(* IEC 61131-3 sources: pandora/pandora/aws-platform-main/aws-platform-main/test/Io, 6 files *)

(* ---- Digital.st ---- *)
USING Esab.Io.Mock;

USING AxUnit;

NAMESPACE Esab.Io.Test

    {TestFixture}
    {Category(IO)}
    CLASS DigitalInputTests
        VAR PRIVATE
            _value : BOOL;
            _input : DigitalInput;
            _changedHandler : DigitalInputChangedListenerMock;
        END_VAR

        {FixtureSetup}
        METHOD PUBLIC TestFixtureSetup
            ;
        END_METHOD

        {TestSetup}
        METHOD PUBLIC TestSetup
            _changedHandler.Id := UINT#0;
            _changedHandler.Value := FALSE;
            // Read two times to reset state.
            _input.Id := UINT#0;
            _input.Read(FALSE);
            _input.Read(FALSE);
        END_METHOD

        {Test}
        METHOD PUBLIC GetValue
            _input.Read(TRUE);
            Assert.Equal(_input.GetValue(), TRUE);
            _input.Read(FALSE);
            Assert.Equal(_input.GetValue(), FALSE);
        END_METHOD

        {Test}
        METHOD PUBLIC RisingEdge
            _input.Read(TRUE);
            Assert.Equal(_input.GetValue(), TRUE);
            Assert.Equal(_input.RisingEdge(), TRUE);
            Assert.Equal(_input.FallingEdge(), FALSE);
            _input.Read(TRUE);
            Assert.Equal(_input.GetValue(), TRUE);
            Assert.Equal(_input.RisingEdge(), FALSE);
            Assert.Equal(_input.FallingEdge(), FALSE);
        END_METHOD

        {Test}
        METHOD PUBLIC FallingEdge
            _input.Read(TRUE);
            Assert.Equal(_input.GetValue(), TRUE);
            _input.Read(FALSE);
            Assert.Equal(_input.GetValue(), FALSE);
            Assert.Equal(_input.RisingEdge(), FALSE);
            Assert.Equal(_input.FallingEdge(), TRUE);
            _input.Read(FALSE);
            Assert.Equal(_input.GetValue(), FALSE);
            Assert.Equal(_input.RisingEdge(), FALSE);
            Assert.Equal(_input.FallingEdge(), FALSE);
        END_METHOD

        {Test}
        METHOD PUBLIC OnChangedRising
            _input.Id := UINT#255;
            _input.SetChangedHandler(_changedHandler);

            _input.Read(FALSE);
            _input.Read(TRUE);

            Assert.Equal(_input.GetValue(), TRUE);
            Assert.Equal(_changedHandler.Id, UINT#255);
            Assert.Equal(_changedHandler.Value, TRUE);
        END_METHOD

        {Test}
        METHOD PUBLIC OnChangedFalling
            _input.Id := UINT#255;
            _input.SetChangedHandler(_changedHandler);

            _input.Read(FALSE);
            _input.Read(TRUE);
            _input.Read(FALSE);

            Assert.Equal(_input.GetValue(), FALSE);
            Assert.Equal(_changedHandler.Id, UINT#255);
            Assert.Equal(_changedHandler.Value, FALSE);
        END_METHOD

        {Test}
        METHOD PUBLIC HasChanged
            _input.Read(TRUE);
            _input.Read(TRUE);
            Assert.Equal(_input.HasChanged(), FALSE);
            _input.Read(FALSE);
            Assert.Equal(_input.HasChanged(), TRUE);
            _input.Read(TRUE);
            Assert.Equal(_input.HasChanged(), TRUE);
        END_METHOD
    END_CLASS

    {TestFixture}
    CLASS DigitalOutputTests
        VAR PRIVATE
            _outputValue : BOOL;
            _output : DigitalOutput;
        END_VAR

        {FixtureSetup}
        METHOD PUBLIC TestFixtureSetup
            ;
        END_METHOD

        {TestSetup}
        METHOD PUBLIC TestSetup
            _outputValue := FALSE;
            _output.SetValue(_outputValue);
        END_METHOD

        {Test}
        METHOD PUBLIC Set
            _output.Set();
            _output.Write(value => _outputValue);

            Assert.Equal(_outputValue, TRUE);
        END_METHOD

        {Test}
        METHOD PUBLIC Reset
            _outputValue := TRUE;
            _output.Reset();
            _output.Write(value => _outputValue);

            Assert.Equal(_outputValue, FALSE);
        END_METHOD

        {Test}
        METHOD PUBLIC Toggle
            _output.Toggle();
            _output.Write(value => _outputValue);

            Assert.Equal(_outputValue, TRUE);

            _output.Toggle();
            _output.Write(value => _outputValue);

            Assert.Equal(_outputValue, FALSE);
        END_METHOD

        {Test}
        METHOD PUBLIC ToggleRepeatedly
            _output.Toggle();
            _output.Toggle();
            _output.Toggle();
            _output.Toggle();
            _output.Toggle();
            _output.Write(value => _outputValue);

            Assert.Equal(_outputValue, TRUE);
            _output.Toggle();
            _output.Toggle();
            _output.Toggle();
            _output.Toggle();
            _output.Toggle();
            _output.Write(value => _outputValue);

            Assert.Equal(_outputValue, FALSE);
        END_METHOD

        {Test}
        METHOD PUBLIC SetValue
            _output.SetValue(TRUE);
            _output.Write(value => _outputValue);

            Assert.Equal(_outputValue, TRUE);

            _output.SetValue(FALSE);
            _output.Write(value => _outputValue);

            Assert.Equal(_outputValue, FALSE);
        END_METHOD
    END_CLASS

    CLASS DigitalInputChangedListenerMock IMPLEMENTS InputChangedListener
        VAR PUBLIC
            Id : UINT;
            Value : BOOL;
        END_VAR

        METHOD PUBLIC InputChanged
            VAR_INPUT
                input : REF_TO Input;
            END_VAR

            VAR_TEMP
                _input : REF_TO DigitalInput;
            END_VAR

            _input ?= input;

            IF _input <> NULL THEN
                Id := _input^.Id;
                Value := _input^.GetValue();
            END_IF;
        END_METHOD
    END_CLASS

END_NAMESPACE

(* ---- DInt.st ---- *)
USING Esab.Io.Mock;

USING AxUnit;

NAMESPACE Esab.Io.Test

    {TestFixture}
    {Category(IO)}
    CLASS DIntInputTests
        VAR PRIVATE
            _value : BOOL;
            _input : DIntInput;
            _changedHandler : DIntInputChangedListenerMock;
        END_VAR

        {FixtureSetup}
        METHOD PUBLIC TestFixtureSetup
            ;
        END_METHOD

        {TestSetup}
        METHOD PUBLIC TestSetup
            _changedHandler.Id := UINT#0;
            _changedHandler.Value := 0;
            _input.Id := UINT#0;
            // Read two times to reset state.
            _input.Endianness := Endianness#Big;
            _input.Read(0);
            _input.Read(0);
        END_METHOD

        {Test}
        METHOD PUBLIC ReadBigEndian
            _input.Read(DINT#16#11121314);
            Assert.Equal(_input.GetValue(), DINT#16#11121314);
            _input.Read(0);
            Assert.Equal(_input.GetValue(), 0);
        END_METHOD

        {Test}
        METHOD PUBLIC ReadLittleEndian
            _input.Endianness := Endianness#Little;
            _input.Read(DINT#16#11121314);
            Assert.Equal(_input.GetValue(), DINT#16#14131211);
            _input.Read(0);
            Assert.Equal(_input.GetValue(), 0);
        END_METHOD

        {Test}
        METHOD PUBLIC GetValue
            _input.Read(25);
            Assert.Equal(_input.GetValue(), 25);
            _input.Read(0);
            Assert.Equal(_input.GetValue(), 0);
        END_METHOD

        {Test}
        METHOD PUBLIC HasChanged
            _input.Read(25);
            Assert.Equal(_input.GetValue(), 25);
            _input.Read(50);
            Assert.Equal(_input.HasChanged(), TRUE);
        END_METHOD

        {Test}
        METHOD PUBLIC OnChanged
            _input.Id := UINT#255;
            _input.SetChangedHandler(_changedHandler);

            _input.Read(0);
            _input.Read(25);

            Assert.Equal(_input.GetValue(), 25);
            Assert.Equal(_changedHandler.Id, UINT#255);
            Assert.Equal(_changedHandler.Value, 25);
        END_METHOD
    END_CLASS

    {TestFixture}
    CLASS DIntOutputTests
        VAR PRIVATE
            _outputValue : DINT;
            _output : DintOutput;
        END_VAR

        {FixtureSetup}
        METHOD PUBLIC TestFixtureSetup
            ;
        END_METHOD

        {TestSetup}
        METHOD PUBLIC TestSetup
            _outputValue := 0;
            _output.Endianness := Endianness#Big;
            _output.SetValue(_outputValue);
        END_METHOD

        {Test}
        METHOD PUBLIC WriteBigEndian
            _output.SetValue(DINT#16#11121314);
            _output.Write(_outputValue);

            Assert.Equal(_outputValue, DINT#16#11121314);
        END_METHOD

        {Test}
        METHOD PUBLIC WriteLittleEndian
            _output.Endianness := Endianness#Little;
            _output.SetValue(DINT#16#11121314);
            _output.Write(_outputValue);

            Assert.Equal(_outputValue, DINT#16#14131211);
        END_METHOD

        {Test}
        METHOD PUBLIC SetValue
            _output.SetValue(25);
            _output.Write(value => _outputValue);

            Assert.Equal(_outputValue, 25);

            _output.SetValue(0);
            _output.Write(value => _outputValue);

            Assert.Equal(_outputValue, 0);
        END_METHOD
    END_CLASS

    CLASS DIntInputChangedListenerMock IMPLEMENTS InputChangedListener
        VAR PUBLIC
            Id : UINT;
            Value : DINT;
        END_VAR

        METHOD PUBLIC InputChanged
            VAR_INPUT
                input : REF_TO Input;
            END_VAR

            VAR_TEMP
                _input : REF_TO DIntInput;
            END_VAR

            _input ?= input;

            IF _input <> NULL THEN
                Id := _input^.Id;
                Value := _input^.GetValue();
            END_IF;
        END_METHOD
    END_CLASS

END_NAMESPACE

(* ---- Int.st ---- *)
USING Esab.Io.Mock;

USING AxUnit;

NAMESPACE Esab.Io.Test

    {TestFixture}
    {Category(IO)}
    CLASS IntInputTests
        VAR PRIVATE
            _value : BOOL;
            _input : IntInput;
            _changedHandler : IntInputChangedListenerMock;
        END_VAR

        {FixtureSetup}
        METHOD PUBLIC TestFixtureSetup
            ;
        END_METHOD

        {TestSetup}
        METHOD PUBLIC TestSetup
            _changedHandler.Id := UINT#0;
            _changedHandler.Value := 0;
            _input.Id := UINT#0;
            // Read two times to reset state.
            _input.Endianness := Endianness#Big;
            _input.Read(0);
            _input.Read(0);
        END_METHOD

        {Test}
        METHOD PUBLIC ReadBigEndian
            _input.Read(16#1216);
            Assert.Equal(_input.GetValue(), 16#1216);
            _input.Read(0);
            Assert.Equal(_input.GetValue(), 0);
        END_METHOD

        {Test}
        METHOD PUBLIC ReadLittleEndian
            _input.Endianness := Endianness#Little;
            _input.Read(16#1216);
            Assert.Equal(_input.GetValue(), 16#1612);
            _input.Read(0);
            Assert.Equal(_input.GetValue(), 0);
        END_METHOD

        {Test}
        METHOD PUBLIC HasChanged
            _input.Read(25);
            Assert.Equal(_input.GetValue(), 25);
            _input.Read(50);
            Assert.Equal(_input.HasChanged(), TRUE);
        END_METHOD

        {Test}
        METHOD PUBLIC OnChanged
            _input.Id := UINT#255;
            _input.SetChangedHandler(_changedHandler);

            _input.Read(0);
            _input.Read(25);

            Assert.Equal(_input.GetValue(), 25);
            Assert.Equal(_changedHandler.Id, UINT#255);
            Assert.Equal(_changedHandler.Value, 25);
        END_METHOD
    END_CLASS

    {TestFixture}
    CLASS IntOutputTests
        VAR PRIVATE
            _outputValue : INT;
            _output : IntOutput;
        END_VAR

        {FixtureSetup}
        METHOD PUBLIC TestFixtureSetup
            ;
        END_METHOD

        {TestSetup}
        METHOD PUBLIC TestSetup
            _outputValue := 0;
            _output.Endianness := Endianness#Big;
            _output.SetValue(_outputValue);
        END_METHOD

        {Test}
        METHOD PUBLIC WriteBigEndian
            _output.SetValue(16#1215);
            _output.Write(_outputValue);

            Assert.Equal(_outputValue, 16#1215);
        END_METHOD

        {Test}
        METHOD PUBLIC WriteLittleEndian
            _output.Endianness := Endianness#Little;
            _output.SetValue(16#1215);
            _output.Write(_outputValue);

            Assert.Equal(_outputValue, 16#1512);
        END_METHOD

        {Test}
        METHOD PUBLIC SetValue
            _output.SetValue(16);
            _output.Write(value => _outputValue);

            Assert.Equal(_outputValue, 16);

            _output.SetValue(0);
            _output.Write(value => _outputValue);

            Assert.Equal(_outputValue, 0);
        END_METHOD
    END_CLASS

    CLASS IntInputChangedListenerMock IMPLEMENTS InputChangedListener
        VAR PUBLIC
            Id : UINT;
            Value : INT;
        END_VAR

        METHOD PUBLIC InputChanged
            VAR_INPUT
                input : REF_TO Input;
            END_VAR

            VAR_TEMP
                _input : REF_TO IntInput;
            END_VAR

            _input ?= input;

            IF _input <> NULL THEN
                Id := _input^.Id;
                Value := _input^.GetValue();
            END_IF;
        END_METHOD
    END_CLASS

END_NAMESPACE

(* ---- Real.st ---- *)
USING Esab.Io.Mock;

USING AxUnit;

NAMESPACE Esab.Io.Test

    {TestFixture}
    {Category(IO)}
    CLASS RealInputTests
        VAR PRIVATE
            _value : BOOL;
            _input : RealInput;
            _changedHandler : RealInputChangedListenerMock;
        END_VAR

        {FixtureSetup}
        METHOD PUBLIC TestFixtureSetup
            ;
        END_METHOD

        {TestSetup}
        METHOD PUBLIC TestSetup
            _changedHandler.Id := UINT#0;
            _changedHandler.Value := 0;
            _input.Id := UINT#0;
            _input.Scale := REAL#1.0;
            _input.Endianness := Endianness#Big;
            // Read two times to reset state.
            _input.Read(0);
            _input.Read(0);
        END_METHOD

        {Test}
        METHOD PUBLIC ReadBigEndian
            _input.Read(DWORD#16#11121314);
            Assert.Equal(TO_DWORD(_input.GetValue()), DWORD#16#11121314);
        END_METHOD

        {Test}
        METHOD PUBLIC ReadLittleEndian
            _input.Endianness := Endianness#Little;
            _input.Read(DWORD#16#11121314);
            Assert.Equal(TO_DWORD(_input.GetValue()), DWORD#16#14131211);
        END_METHOD

        {Test}
        METHOD PUBLIC ReadRealWithScaling
            _input.Scale := REAL#0.01;
            _input.Read(REAL#100.0);
            Assert.InRange(_input.GetValue(), REAL#1.0, REAL#0.001);
        END_METHOD

        {Test}
        METHOD PUBLIC ReadDwordWithScaling
            _input.Scale := REAL#0.01;
            _input.Read(TO_DWORD(REAL#100.0));
            Assert.InRange(_input.GetValue(), REAL#1.0, REAL#0.001);
        END_METHOD

        {Test}
        METHOD PUBLIC ReadUIntWithScaling
            _input.Scale := REAL#0.01;
            _input.Read(UINT#100);
            Assert.InRange(_input.GetValue(), REAL#1.0, REAL#0.001);
        END_METHOD

        {Test}
        METHOD PUBLIC ReadIntWithScaling
            _input.Scale := REAL#0.01;
            _input.Read(INT#100);
            Assert.InRange(_input.GetValue(), REAL#1.0, REAL#0.001);
        END_METHOD

        {Test}
        METHOD PUBLIC HasChanged
            _input.Read(25);
            Assert.Equal(_input.GetValue(), 25);
            _input.Read(50);
            Assert.Equal(_input.HasChanged(), TRUE);
        END_METHOD

        {Test}
        METHOD PUBLIC OnChanged
            _input.Id := UINT#255;
            _input.SetChangedHandler(_changedHandler);

            _input.Read(0);
            _input.Read(25);

            Assert.Equal(_input.GetValue(), 25);
            Assert.Equal(_changedHandler.Id, UINT#255);
            Assert.Equal(_changedHandler.Value, 25);
        END_METHOD
    END_CLASS

    {TestFixture}
    {Category(IO)}
    CLASS RealOutputTests
        VAR PRIVATE
            _outputValue : REAL;
            _output : RealOutput;
        END_VAR

        {FixtureSetup}
        METHOD PUBLIC TestFixtureSetup
            ;
        END_METHOD

        {TestSetup}
        METHOD PUBLIC TestSetup
            _outputValue := 0;
            _output.Scale := REAL#1.0;
            _output.Endianness := Endianness#Big;
            _output.SetValue(_outputValue);
        END_METHOD

        {Test}
        METHOD PUBLIC WriteBigEndian
            _output.SetValue(TO_REAL(DWORD#16#11121314));
            _output.Write(_outputValue);
            Assert.Equal(_outputValue, TO_REAL(DWORD#16#11121314));
        END_METHOD

        {Test}
        METHOD PUBLIC WriteLittleEndian
            _output.Endianness := Endianness#Little;
            _output.SetValue(TO_REAL(DWORD#16#11121314));
            _output.Write(_outputValue);

            Assert.Equal(_outputValue, TO_REAL(DWORD#16#14131211));
        END_METHOD

        {Test}
        METHOD PUBLIC WriteRealWithScaling
            VAR_TEMP
                value : REAL;
            END_VAR

            _output.Scale := REAL#0.01;
            _output.SetValue(REAL#3.14);
            _output.Write(value);
            Assert.InRange(value, REAL#314.0, REAL#0.001);
        END_METHOD

        {Test}
        METHOD PUBLIC WriteDWordWithScaling
            VAR_TEMP
                value : DWORD;
            END_VAR

            _output.Scale := REAL#0.01;
            _output.SetValue(REAL#3.14);
            _output.Write(value);
            Assert.InRange(TO_REAL(value), REAL#314.0, REAL#0.001);
        END_METHOD

        {Test}
        METHOD PUBLIC WriteUIntWithScaling
            VAR_TEMP
                value : UINT;
            END_VAR

            _output.Scale := REAL#0.01;
            _output.SetValue(REAL#3.14);
            _output.Write(value);
            Assert.Equal(value, UINT#314);
        END_METHOD

        {Test}
        METHOD PUBLIC WriteIntWithScaling
            VAR_TEMP
                value : INT;
            END_VAR

            _output.Scale := REAL#0.01;
            _output.SetValue(REAL#3.14);
            _output.Write(value);
            Assert.Equal(value, INT#314);
        END_METHOD

        {Test}
        METHOD PUBLIC SetValue
            _output.SetValue(16);
            _output.Write(value => _outputValue);

            Assert.Equal(_outputValue, 16);

            _output.SetValue(0);
            _output.Write(value => _outputValue);

            Assert.Equal(_outputValue, 0);
        END_METHOD
    END_CLASS

    {TestFixture}
    {Category(IO)}
    CLASS RealNormalizedInputTests
        VAR PRIVATE
            _inputValue : REAL;
            _input : RealNormalizedInput;
        END_VAR

        {FixtureSetup}
        METHOD PUBLIC TestFixtureSetup
            ;
        END_METHOD

        {TestSetup}
        METHOD PUBLIC TestSetup
            _inputValue := 0;
            _input.Endianness := Endianness#Big;
            _input.Bipolar := FALSE;
            _input.Minimum := REAL#0.0;
            _input.Maximum := REAL#27648.0;
            _input.Read(_inputValue);
        END_METHOD

        {Test}
        METHOD PUBLIC ReadNormalizedWithDefaults
            _input.Read(27648);

            _inputValue := _input.GetValue();

            Assert.InRange(_inputValue, 1.0, 0.001);

            _input.Read(13824);

            _inputValue := _input.GetValue();

            Assert.InRange(_inputValue, 0.5, 0.001);

            _input.Read(0);

            _inputValue := _input.GetValue();

            Assert.InRange(_inputValue, 0.0, 0.001);
        END_METHOD

        {Test}
        METHOD PUBLIC ReadNormalizedBipolar
            _input.Bipolar := TRUE;
            _input.Minimum := -REAL#27648.0;
            _input.Maximum := REAL#27648.0;

            _input.Read(27648);

            _inputValue := _input.GetValue();

            Assert.InRange(_inputValue, 1.0, 0.001);

            _input.Read(0);

            _inputValue := _input.GetValue();

            Assert.InRange(_inputValue, 0.0, 0.001);

            _input.Read(-27648);

            _inputValue := _input.GetValue();

            Assert.InRange(_inputValue, -1.0, 0.001);
        END_METHOD
    END_CLASS

    {TestFixture}
    {Category(IO)}
    CLASS RealNormalizedOutputTests
        VAR PRIVATE
            _outputValue : INT;
            _output : RealNormalizedOutput;
        END_VAR

        {FixtureSetup}
        METHOD PUBLIC TestFixtureSetup
            ;
        END_METHOD

        {TestSetup}
        METHOD PUBLIC TestSetup
            _outputValue := 0;
            _output.Endianness := Endianness#Big;
            _output.Bipolar := FALSE;
            _output.Minimum := REAL#0.0;
            _output.Maximum := REAL#27648.0;
            _output.SetValue(0);
        END_METHOD

        {Test}
        METHOD PUBLIC WriteNormalizedWithDefaults
            _output.SetValue(REAL#1.0);
            _output.Write(_outputValue);
            Assert.InRange(_outputValue, 27648, 0.001);

            _output.SetValue(REAL#0.5);
            _output.Write(_outputValue);
            Assert.InRange(_outputValue, 27648/2, 0.001);

            _output.SetValue(REAL#0.0);
            _output.Write(_outputValue);
            Assert.InRange(_outputValue, 0, 0.001);
        END_METHOD

        {Test}
        METHOD PUBLIC WriteNormalizedBipolar
            _output.Bipolar := TRUE;
            _output.Minimum := -REAL#27648.0;
            _output.Maximum := REAL#27648.0;

            _output.SetValue(REAL#1.0);
            _output.Write(_outputValue);
            Assert.InRange(_outputValue, 27648, 0.001);

            _output.SetValue(REAL#0.5);
            _output.Write(_outputValue);
            Assert.InRange(_outputValue, 27648/2, 0.001);

            _output.SetValue(REAL#0.0);
            _output.Write(_outputValue);
            Assert.InRange(_outputValue, 0, 0.001);

            _output.SetValue(REAL#-0.5);
            _output.Write(_outputValue);
            Assert.InRange(_outputValue, -27648/2, 0.001);

            _output.SetValue(REAL#-1.0);
            _output.Write(_outputValue);
            Assert.InRange(_outputValue, -27648, 0.001);
        END_METHOD

        {Test}
        METHOD PUBLIC WriteLargerThan1
            _output.SetValue(REAL#10.0);
            _output.Write(_outputValue);
            Assert.InRange(_outputValue, 27648, 0.001);
        END_METHOD
    END_CLASS

    CLASS RealInputChangedListenerMock IMPLEMENTS InputChangedListener
        VAR PUBLIC
            Id : UINT;
            Value : REAL;
        END_VAR

        METHOD PUBLIC InputChanged
            VAR_INPUT
                input : REF_TO Input;
            END_VAR

            VAR_TEMP
                _input : REF_TO RealInput;
            END_VAR

            _input ?= input;

            IF _input <> NULL THEN
                Id := _input^.Id;
                Value := _input^.GetValue();
            END_IF;
        END_METHOD
    END_CLASS

END_NAMESPACE

(* ---- UInt.st ---- *)
USING Esab.Io.Mock;

USING AxUnit;

NAMESPACE Esab.Io.Test

    {TestFixture}
    {Category(IO)}
    CLASS UIntInputTests
        VAR PRIVATE
            _value : BOOL;
            _input : UIntInput;
            _listener : UIntInputChangedListenerMock;
        END_VAR

        {FixtureSetup}
        METHOD PUBLIC TestFixtureSetup
            ;
        END_METHOD

        {TestSetup}
        METHOD PUBLIC TestSetup
            _listener.Id := UINT#0;
            _listener.Value := UINT#0;
            _input.Id := UINT#0;
            // Read two times to reset state.
            _input.Endianness := Endianness#Big;
            _input.Read(UINT#0);
            _input.Read(UINT#0);
        END_METHOD

        {Test}
        METHOD PUBLIC ReadBigEndian
            _input.Read(UINT#16#1216);
            Assert.Equal(_input.GetValue(), UINT#16#1216);
        END_METHOD

        {Test}
        METHOD PUBLIC ReadLittleEndian
            _input.Endianness := Endianness#Little;
            _input.Read(UINT#16#1216);
            Assert.Equal(_input.GetValue(), UINT#16#1612);
        END_METHOD

        {Test}
        METHOD PUBLIC ReadBigEndianByte
            _input.Read(BYTE#16#16);
            Assert.Equal(_input.GetValue(), UINT#16#16);
        END_METHOD

        {Test}
        METHOD PUBLIC ReadLittleEndianByte
            _input.Endianness := Endianness#Little;
            _input.Read(BYTE#16#16);
            Assert.Equal(_input.GetValue(), UINT#16#16);
        END_METHOD

        {Test}
        METHOD PUBLIC HasChanged
            _input.Read(UINT#25);
            Assert.Equal(_input.GetValue(), UINT#25);
            _input.Read(UINT#50);
            Assert.Equal(_input.HasChanged(), TRUE);
        END_METHOD

        {Test}
        METHOD PUBLIC OnChanged
            _input.Id := UINT#255;
            _input.SetChangedHandler(_listener);

            _input.Read(UINT#0);
            _input.Read(UINT#25);

            Assert.Equal(_input.GetValue(), UINT#25);
            Assert.Equal(_listener.Id, UINT#255);
            Assert.Equal(_listener.Value, UINT#25);
        END_METHOD
    END_CLASS

    {TestFixture}
    CLASS UIntOutputTests
        VAR PRIVATE
            _outputValue : UINT;
            _output : UIntOutput;
        END_VAR

        {FixtureSetup}
        METHOD PUBLIC TestFixtureSetup
            ;
        END_METHOD

        {TestSetup}
        METHOD PUBLIC TestSetup
            _outputValue := UINT#0;
            _output.Endianness := Endianness#Big;
            _output.SetValue(_outputValue);
        END_METHOD

        {Test}
        METHOD PUBLIC WriteBigEndian
            _output.SetValue(UINT#16#1215);
            _output.Write(_outputValue);

            Assert.Equal(_outputValue, UINT#16#1215);
        END_METHOD

        {Test}
        METHOD PUBLIC WriteLittleEndian
            _output.Endianness := Endianness#Little;
            _output.SetValue(UINT#16#1215);
            _output.Write(_outputValue);

            Assert.Equal(_outputValue, UINT#16#1512);
        END_METHOD

        {Test}
        METHOD PUBLIC WriteBigEndianByte
            VAR_TEMP
                b : BYTE;
            END_VAR

            _output.SetValue(UINT#16#1215);
            _output.Write(b);

            Assert.Equal(b, BYTE#16#15);
        END_METHOD

        {Test}
        METHOD PUBLIC WriteLittleEndianByte
            VAR_TEMP
                b : BYTE;
            END_VAR

            _output.SetValue(UINT#16#1215);
            _output.Write(b);

            Assert.Equal(b, BYTE#16#15);
        END_METHOD

        {Test}
        METHOD PUBLIC SetValue
            _output.SetValue(UINT#16);
            _output.Write(value => _outputValue);

            Assert.Equal(_outputValue, UINT#16);

            _output.SetValue(UINT#0);
            _output.Write(value => _outputValue);

            Assert.Equal(_outputValue, UINT#0);
        END_METHOD
    END_CLASS

    CLASS UIntInputChangedListenerMock IMPLEMENTS InputChangedListener
        VAR PUBLIC
            Id : UINT;
            Value : UINT;
        END_VAR

        METHOD PUBLIC InputChanged
            VAR_INPUT
                input : REF_TO Input;
            END_VAR

            VAR_TEMP
                _input : REF_TO UIntInput;
            END_VAR

            _input ?= input;

            IF _input <> NULL THEN
                Id := _input^.Id;
                Value := _input^.GetValue();
            END_IF;
        END_METHOD
    END_CLASS

END_NAMESPACE

(* ---- Word.st ---- *)
USING Esab.Io.Mock;

USING AxUnit;

NAMESPACE Esab.Io.Test

    {TestFixture}
    {Category(IO)}
    CLASS WordInputTests
        VAR PRIVATE
            _value : BOOL;
            _input : WordInput;
            _listener : WordInputChangedListenerMock;
        END_VAR

        {FixtureSetup}
        METHOD PUBLIC TestFixtureSetup
            ;
        END_METHOD

        {TestSetup}
        METHOD PUBLIC TestSetup
            _listener.Id := UINT#0;
            _listener.Value := WORD#0;
            _input.Id := UINT#0;
            // Read two times to reset state.
            _input.Endianness := Endianness#Big;
            _input.Read(WORD#0);
            _input.Read(WORD#0);
        END_METHOD

        {Test}
        METHOD PUBLIC ReadBigEndian
            _input.Read(WORD#16#1216);
            Assert.Equal(_input.GetValue(), WORD#16#1216);
        END_METHOD

        {Test}
        METHOD PUBLIC ReadLittleEndian
            _input.Endianness := Endianness#Little;
            _input.Read(WORD#16#1216);
            Assert.Equal(_input.GetValue(), WORD#16#1612);
        END_METHOD

        {Test}
        METHOD PUBLIC ReadBigEndianByte
            _input.Read(BYTE#16#16);
            Assert.Equal(_input.GetValue(), WORD#16#16);
        END_METHOD

        {Test}
        METHOD PUBLIC ReadLittleEndianByte
            _input.Endianness := Endianness#Little;
            _input.Read(BYTE#16#16);
            Assert.Equal(_input.GetValue(), WORD#16#16);
        END_METHOD

        {Test}
        METHOD PUBLIC HasChanged
            _input.Read(WORD#25);
            Assert.Equal(_input.GetValue(), WORD#25);
            _input.Read(WORD#50);
            Assert.Equal(_input.HasChanged(), TRUE);
        END_METHOD

        {Test}
        METHOD PUBLIC OnChanged
            _input.Id := UINT#255;
            _input.SetChangedHandler(_listener);

            _input.Read(WORD#0);
            _input.Read(WORD#25);

            Assert.Equal(_input.GetValue(), WORD#25);
            Assert.Equal(_listener.Id, UINT#255);
            Assert.Equal(_listener.Value, WORD#25);
        END_METHOD
    END_CLASS

    {TestFixture}
    CLASS WordOutputTests
        VAR PRIVATE
            _outputValue : WORD;
            _output : WordOutput;
        END_VAR

        {FixtureSetup}
        METHOD PUBLIC TestFixtureSetup
            ;
        END_METHOD

        {TestSetup}
        METHOD PUBLIC TestSetup
            _outputValue := WORD#0;
            _output.Endianness := Endianness#Big;
            _output.SetValue(_outputValue);
        END_METHOD

        {Test}
        METHOD PUBLIC WriteBigEndian
            _output.SetValue(WORD#16#1215);
            _output.Write(_outputValue);

            Assert.Equal(_outputValue, WORD#16#1215);
        END_METHOD

        {Test}
        METHOD PUBLIC WriteLittleEndian
            _output.Endianness := Endianness#Little;
            _output.SetValue(WORD#16#1215);
            _output.Write(_outputValue);

            Assert.Equal(_outputValue, WORD#16#1512);
        END_METHOD

        {Test}
        METHOD PUBLIC WriteBigEndianByte
            VAR_TEMP
                b : BYTE;
            END_VAR

            _output.SetValue(WORD#16#1215);
            _output.Write(b);

            Assert.Equal(b, BYTE#16#15);
        END_METHOD

        {Test}
        METHOD PUBLIC WriteLittleEndianByte
            VAR_TEMP
                b : BYTE;
            END_VAR

            _output.SetValue(WORD#16#1215);
            _output.Write(b);

            Assert.Equal(b, BYTE#16#15);
        END_METHOD

        {Test}
        METHOD PUBLIC SetValue
            _output.SetValue(WORD#16);
            _output.Write(value => _outputValue);

            Assert.Equal(_outputValue, WORD#16);

            _output.SetValue(WORD#0);
            _output.Write(value => _outputValue);

            Assert.Equal(_outputValue, WORD#0);
        END_METHOD

        {Test}
        METHOD PUBLIC SetValueByte
            _output.SetValue(BYTE#127);
            _output.Write(value => _outputValue);

            Assert.Equal(_outputValue, WORD#127);

            _output.SetValue(BYTE#0);
            _output.Write(value => _outputValue);

            Assert.Equal(_outputValue, WORD#0);
        END_METHOD
    END_CLASS

    CLASS WordInputChangedListenerMock IMPLEMENTS InputChangedListener
        VAR PUBLIC
            Id : UINT;
            Value : WORD;
        END_VAR

        METHOD PUBLIC InputChanged
            VAR_INPUT
                input : REF_TO Input;
            END_VAR

            VAR_TEMP
                _input : REF_TO WordInput;
            END_VAR

            _input ?= input;

            IF _input <> NULL THEN
                Id := _input^.Id;
                Value := _input^.GetValue();
            END_IF;
        END_METHOD
    END_CLASS

END_NAMESPACE
